Xinje XCPPro project, PLC1: XC3-32 (software 3.3q)

PROGRAM Ladder

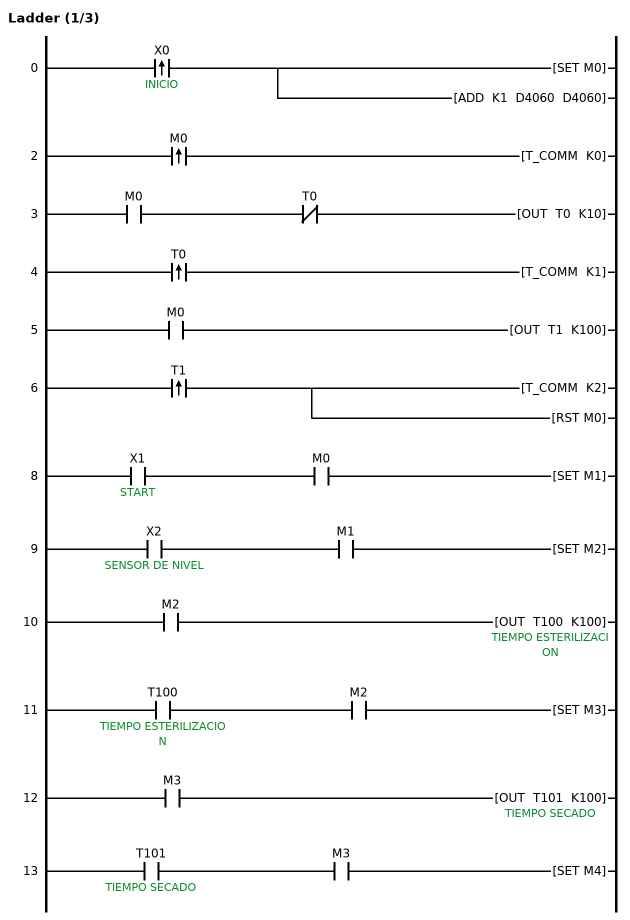
LDP    X0	; INICIO
SET    M0
ADD    K1 D4060 D4060
LDP    M0
T_COMM K0
LD     M0
ANI    T0
OUT    T0 K10
LDP    T0
T_COMM K1
LD     M0
OUT    T1 K100
LDP    T1
T_COMM K2
RST    M0
LD     X1	; START
AND    M0
SET    M1
LD     X2	; SENSOR DE NIVEL
AND    M1
SET    M2
LD     M2
OUT    T100 K100	; TIEMPO ESTERILIZACION
LD     T100	; TIEMPO ESTERILIZACION
AND    M2
SET    M3
LD     M3
OUT    T101 K100	; TIEMPO SECADO
LD     T101	; TIEMPO SECADO
AND    M3
SET    M4

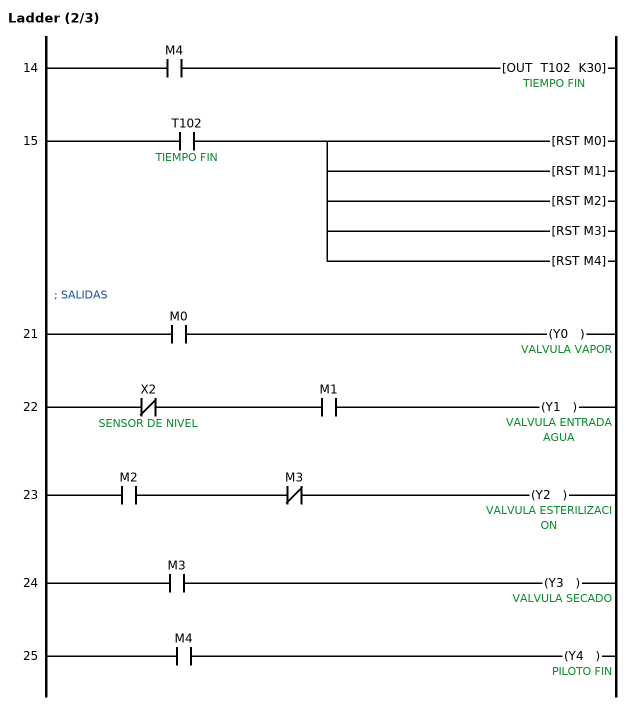
LD     M4
OUT    T102 K30	; TIEMPO FIN
LD     T102	; TIEMPO FIN
RST    M0
RST    M1
RST    M2
RST    M3
RST    M4
; SALIDAS
LD     M0
OUT    Y0	; VALVULA VAPOR
LDI    X2	; SENSOR DE NIVEL
AND    M1
OUT    Y1	; VALVULA ENTRADA AGUA
LD     M2
ANI    M3
OUT    Y2	; VALVULA ESTERILIZACION
LD     M3
OUT    Y3	; VALVULA SECADO
LD     M4
OUT    Y4	; PILOTO FIN

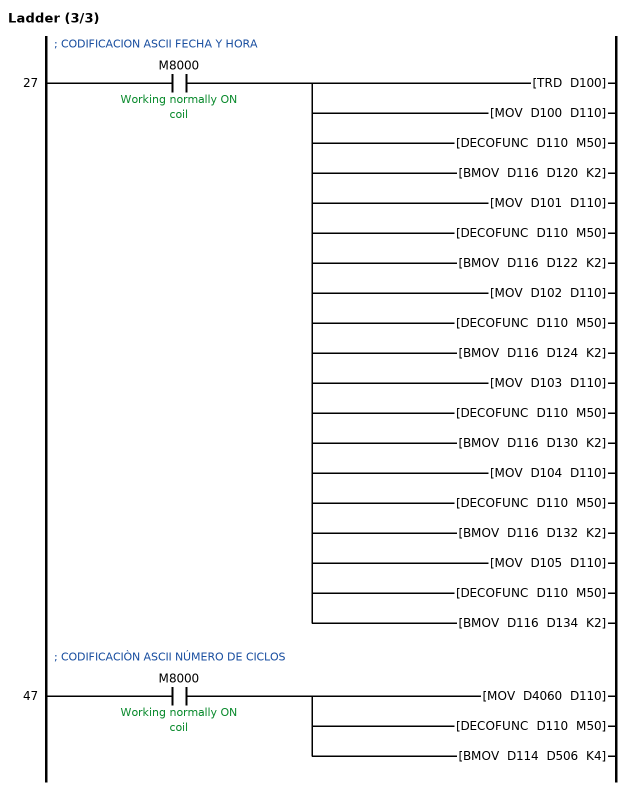
; CODIFICACION ASCII FECHA Y HORA
LD     M8000	; Working normally ON coil
TRD    D100
MOV    D100 D110
DECOFUNC D110 M50
BMOV   D116 D120 K2
MOV    D101 D110
DECOFUNC D110 M50
BMOV   D116 D122 K2
MOV    D102 D110
DECOFUNC D110 M50
BMOV   D116 D124 K2
MOV    D103 D110
DECOFUNC D110 M50
BMOV   D116 D130 K2
MOV    D104 D110
DECOFUNC D110 M50
BMOV   D116 D132 K2
MOV    D105 D110
DECOFUNC D110 M50
BMOV   D116 D134 K2
;  CODIFICACIÒN ASCII NÚMERO DE CICLOS
LD     M8000	; Working normally ON coil
MOV    D4060 D110
DECOFUNC D110 M50
BMOV   D114 D506 K4

CONFIG BLOCK T_COMM K0	; Header
  IsUserInst=false, Inst=SEND, PLCAddr=D1000, ComNum=K2, BufferCount=8, Type=Const, Data="FECHA: ", RegByteCount=0, Type=Reg, Reg=D124, RegByteCount=1, Type=Reg, Reg=D125, RegByteCount=1, Type=Const, Data="/", RegByteCount=0, Type=Reg, Reg=D122, RegByteCount=1, Type=Reg, Reg=D123, RegByteCount=1, Type=Const, Data="/", RegByteCount=0, Type=Reg, Reg=D120, RegByteCount=1, Type=Reg, Reg=D121, RegByteCount=1, Type=Const, Data=13, RegByteCount=0, Type=Const, Data="HORA INICIO: ", RegByteCount=0, Type=Reg, Reg=D130, RegByteCount=1, Type=Reg, Reg=D131, RegByteCount=1, Type=Const, Data=":", RegByteCount=0, Type=Reg, Reg=D132, RegByteCount=1, Type=Reg, Reg=D133, RegByteCount=1, Type=Const, Data=":", RegByteCount=0, Type=Reg, Reg=D134, RegByteCount=1

CONFIG BLOCK T_COMM K1	; Print 1 min
  IsUserInst=false, Inst=SEND, PLCAddr=D1650, ComNum=K2, BufferCount=8, Type=Const, Data="TEMP: ", RegByteCount=0, Type=Const, Data="25 ", RegByteCount=0, Type=Const, Data=248, RegByteCount=0, Type=Const, Data="C ", RegByteCount=0, Type=Const, Data="P: ", RegByteCount=0, Type=Const, Data="110 kpa", RegByteCount=0, Type=Const, Data=13, RegByteCount=0, GUID=ccc18f11-6899-4567-b5f8-e63047ce6ffa

CONFIG BLOCK T_COMM K2	; Footer
  IsUserInst=false, Inst=SEND, PLCAddr=D2000, ComNum=K2, BufferCount=8, Type=Const, Data="HORA FIN: ", RegByteCount=0, Type=Const, Data="13:23:23", RegByteCount=0, Type=Const, Data=13, RegByteCount=0, Type=Const, Data="CICLO COMPLETO", RegByteCount=0, Type=Const, Data=13, RegByteCount=0, Type=Const, Data="Duración: ", RegByteCount=0, Type=Const, Data="38 min", RegByteCount=0, Type=Const, Data=13, RegByteCount=0, Type=Const, Data="DESCARGA: ______________", RegByteCount=0, Type=Const, Data=13, RegByteCount=0, GUID=f6962d61-7d1e-4758-98e8-5b93981797a8

C FUNCTION BLOCK DECOFUNC.FCB
/*************************************************************************
   FunctionBlockName:  DECOFUNC
   Version:            1.0.0
   Author:             
   UpdateTime:         6/12/2023 3:23:16 p. m.
   Comment:            
			
**************************************************************************/
void DECOFUNC( WORD W , BIT B )
{
int data, und, dec, cen, deci, data_raw, temp1, temp2;

data_raw = W[0];

data = abs(data_raw);

if (data >= 1000){
deci = data%10;
temp1 = data/10;
und = temp1%10;
temp2 = temp1/10;
dec = temp2%10;
cen = temp2/10;

W[7] = deci | 0x30;
W[6] = und | 0x30;
W[5] = dec| 0x30;
W[4] = cen | 0x30;

}

if(data >= 100 && data<1000){
und = data%10;
temp1 = data/10;
dec = temp1%10;
cen = temp1/10;

W[4] = 00; //NULL
W[7] = und | 0x30;
W[6] = dec| 0x30;
W[5] = cen | 0x30;
}

if(data >= 10 && data <100 ){
und = data%10;
temp1 = data/10;
dec = temp1%10;

W[5] = 00; //NULL
W[7] = und | 0x30;
W[6] = dec| 0x30;  
W[4] = 00; //NULL

}
if(data >= 0 && data <10 ){
und = data%10;
temp1 = data/10;
W[5] = 00; //NULL
W[7] = und | 0x30;
W[6] = 48; //cero
W[4] = 00; //NULL

}
}